FUNCTION_BLOCK FB_MachineControl_Subsystem
VAR_INPUT
	pMachineCurrentStatus	:POINTER TO E_PMLState;
END_VAR
VAR_OUTPUT
END_VAR
VAR
	machine_status AT%Q*: MachineStatus:= MachineStatus.STOPPED;	
	machine_current_status	: E_PMLState;	
    machineControlCmd	: MachineCommandStructure;
	
	

	bStart	: BOOL;
	bStop	: BOOL;
	bReset	: BOOL;
	machineControlCmd_temp	: MachineCommandStructure;
	AAA: INT;
END_VAR


CASE pMachineCurrentStatus^ OF
	ePMLState_Stopped:
		machine_status	:= MachineStatus.STOPPED;
	ePMLState_Resetting:	
		machine_status	:= MachineStatus.RESETTING;
	ePMLState_Idle:	
		machine_status	:= MachineStatus.READY;	
	ePMLState_Starting:	
		machine_status	:= MachineStatus.INITIALIZING;
	ePMLState_Execute:	
		machine_status	:= MachineStatus.RUNNING;		
	ePMLState_Stopping:	
		machine_status	:= MachineStatus.STOPPING;
	ePMLState_Aborted,ePMLState_Aborting:
		machine_status	:= MachineStatus.ERROR;		
END_CASE




IF bStart THEN
	machineControlCmd_temp.command	:= MachineControlCommand.START;
	machine_control_command(command_data:=machineControlCmd_temp);
	bStart	:= FALSE;
END_IF
IF bStop THEN
	machineControlCmd_temp.command	:= MachineControlCommand.STOP;
	machine_control_command(command_data:=machineControlCmd_temp);
	bStop	:= FALSE;
END_IF
IF bReset THEN
	machineControlCmd_temp.command	:= MachineControlCommand.RESET;
	machine_control_command(command_data:=machineControlCmd_temp);
	bReset	:= FALSE;
END_IF

{attribute 'TcRpcEnable'}
METHOD machine_control_command : UDINT
VAR_INPUT
	command_data : MachineCommandStructure; 	
END_VAR

machineControlCmd	:= command_data;
AAA:=AAA+1;
END_METHOD

END_FUNCTION_BLOCK

(* stored: Version 1.1.0.1, ProductVersion 3.1.4024.12
   POU FB_MachineControl_Subsystem: Id {15e4ff61-708d-44b2-875f-d4ee1da239ec}, SpecialFunc None
   Method machine_control_command: Id {27ade1f0-fc07-41bd-b30c-f2e581ef73ab} *)
